Fanuc KAREL source: kt00505.KL

-- PROVISIONAL review KL for V770-1; original PC SHA256 30dcec8845cd0a384de00ca52b541383587d1d9d109d3817336f001562c65313
-- Incomplete behavior may be omitted. Consult companion uncertainty JSON. Do not deploy.
PROGRAM KT00505
%NOLOCKGROUP
-- UNRESOLVED_DECL P1 type=000102
-- UNRESOLVED_DECL P2 type=000106
-- UNRESOLVED_DECL OUT type=000102
BEGIN
  -- UNRESOLVED_PC offsets 5-20; opcodes 2E,22,32,35
  -- UNRESOLVED_PC offsets 25-40; opcodes 2E,22,32,35
  -- UNRESOLVED_PC offsets 45-84; opcodes 49,7E,49,7E,60,7E,4A
  -- UNRESOLVED_PC offsets 89-93; opcodes 7F
END KT00505
